FUNCTION_BLOCK C_DELAY (* Clocked delayed propagation of an event-Cancellable *)
  (* Standard: 61499-1; Classification: Event processing *)
  (* Version 0.0, 2004-09-23, JHC, Rockwell Automation, SRC version *)
  (* Compiler header: package fb.rt.mva; *)
  (* Compiler Java Sun JDK 1.4.2 *)
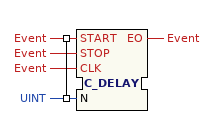
  EVENT_INPUT
    START WITH N; (* Begin Delay *)
    STOP; (* Cancel Delay *)
    CLK; (* Simulation Clock *)
  END_EVENT
  EVENT_OUTPUT
    EO; (* Delayed Event *)
  END_EVENT
  VAR_INPUT
    N : UINT; (* Delay Time in Clock Cycles *)
  END_VAR
  VAR
    COUNT : UINT;
  END_VAR
  ALGORITHM START IN Java: (* Initialization algorithm *)
if(COUNT.value==0) COUNT.value = N.value;
  END_ALGORITHM
  ALGORITHM STOP IN Java: (* Normally executed algorithm *)
COUNT.value=0;
  END_ALGORITHM
  ALGORITHM CLK IN Java: (* Normally executed algorithm *)
if(COUNT.value==0) return;
COUNT.value--;
if(COUNT.value==0) EO.serviceEvent(this);
  END_ALGORITHM
END_FUNCTION_BLOCK
